TYPE
    ST_Detail_Descriptions : STRUCT
        Detail_Key : ARRAY[1..Global.MAX_DETAIL_COUNT] OF ST_KeyValue;
    END_STRUCT
END_TYPE

(* stored: Version 1.1.0.1
   DUT ST_Detail_Descriptions: Id {7f285689-5356-4ebc-b14c-cf1c1063e295} *)
